TYPE teCTCBrakeMode :
(
	CTC_BRAKE_MODE_OFF := 0,
	CTC_BRAKE_MODE_WHEN_DISABLED := 1,
	CTC_BRAKE_MODE_IN_STANDSTILL := 2
);
END_TYPE

(* stored: Version 1.1.0.1, ProductVersion 3.1.4026.17
   EnumerationTextList teCTCBrakeMode: Id {58873ecb-6c45-4d9c-a1c2-66f49aef99d0} *)
